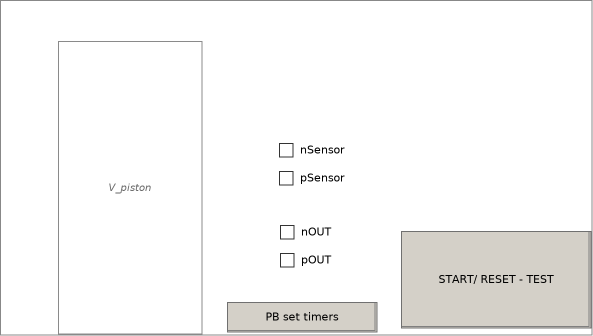
VISUALIZATION Visualization  // 593x336
    Frame (58,41 144x293)
        shows V_piston(p := MAIN.p1)
    Checkbox (277,135 150x30), "nSensor", variable: MAIN.nSensor
    Checkbox (277,163 150x30), "pSensor", variable: MAIN.pSensor
    Checkbox (278,217 150x30), "nOUT", variable: MAIN.nOut
    Checkbox (278,245 150x30), "pOUT", variable: MAIN.pOut
    Button (227,302 150x30), "PB set timers"
        OnMouseDown: execute { main.pbSetTimers := TRUE; }
        OnMouseUp: execute { main.pbSetTimers := FALSE; }
    Button (401,231 190x97), "START/ RESET - TEST"
        OnMouseDown: execute { main.PB := TRUE; }
        OnMouseUp: execute { main.PB := FALSE; }
END_VISUALIZATION

(* stored: Version 1.1.0.1, ProductVersion 3.1.4022.18
   Visu Visualization: Id {ed9e1219-b857-432c-86ff-b28175938f1e} *)
